{attribute 'linkalways'} 
{attribute 'no_explicit_call' := 'This FB is a CLASS and must be accessed using methods or properties'}
{attribute 'enable_dynamic_creation'}
FUNCTION_BLOCK Node_F_VN_CountNonZeroPixels EXTENDS VisionNode
VAR
    ipSrcImage : _ITcVnImage;
    nNonZero : _ULINT(0);
    hrPrev : _HRESULT(S_OK);
	hresult : _HRESULT(S_OK);
END_VAR

METHOD PUBLIC  Clone : I_Node
VAR
	pNode : POINTER TO Node_F_VN_CountNonZeroPixels;
END_VAR
pNode := __NEW(Node_F_VN_CountNonZeroPixels);
Clone := pNode^;
END_METHOD

METHOD FB_init : BOOL
VAR_INPUT
	bInitRetains : BOOL; // if TRUE, the retain variables are initialized (warm start / cold start)
	bInCopyCode : BOOL;  // if TRUE, the instance afterwards gets moved into the copy code (online change)
END_VAR
AddInput('ipSrcImage', ipSrcImage);
AddInput('hrPrev', hrPrev);
AddOutput('nNonZero', nNonZero);
AddOutput('hresult', hresult);
END_METHOD

METHOD PROTECTED  OnExecute : HRESULT
hresult.Value := F_VN_CountNonZeroPixels(
	ipSrcImage := ipSrcImage.Value,
    nNonZero := nNonZero.Value,
	hrPrev:= hrPrev.Value);
END_METHOD

METHOD PUBLIC PreExecutionCheck
VAR_INPUT
	Check : I_PreExecutionChecks;
END_VAR
Check.IsTrue(ipSrcImage.IsValid, 'ipSrcImage must contain an image');
Check.IsTrue(ipSrcImage.HasChannelCount(1), 'ipSrcImage must contain 1 channel');
END_METHOD

END_FUNCTION_BLOCK

(* stored: Version 1.1.0.1, ProductVersion 3.1.4024.13
   POU Node_F_VN_CountNonZeroPixels: Id {d7d6579d-a94a-0100-27a7-ffbccb677052}, SpecialFunc None
   Folder Constructor: Id {664a347a-d6c7-0d67-3a4b-3c65e07d20b4}
   Method Clone: Id {11087c25-fdf9-055a-2d95-6e724a0a2387}
   Method FB_init: Id {52aafdc6-5ff7-0163-2410-45217f423104}
   Method OnExecute: Id {e369dc1b-5f6d-0828-377e-9b9ea2b9c609}
   Method PreExecutionCheck: Id {1ac31727-e972-0f99-07ac-ce45971424de} *)
